Staubli VAL3: onStart.pgx

program onStart()
  local num i
  local string l_sMessage
  local string l_sPath
  local num l_nResult
begin
  // INIT
  sPath=""
  bExit=false
  nIndex=nSelected=nView=nId=0
  // reset the Key pressure
  call use:nullKey(nKey)
  // logMsg
  logMsg("[KERNEL] INTERFACE:PAGE edit program")
  // load the program TYPE
  call saveData:getPathInstr(saveData:sProgTypeUsing,l_sPath)
  l_nResult=prog:libLoad(l_sPath)
  delay(0)
  // program name
  sProgram=sItems[0]
  call prog:load(sProgram,i)
  //
  if i!=0
    call language:message(l_sMessage,-7)
    popUpMsg(l_sMessage+" PROG "+sProgram+" code "+toString("",i))
  endIf
  // unselect ALL
  call prog:unSelectItem()
  // define the list
  call buildList()
  // build the page
  call refreshStatic()
end
